FUNCTION_BLOCK Queue
VAR_INPUT
END_VAR
VAR_OUTPUT
END_VAR
VAR
	bAddTailValue		: BOOL := TRUE;
	bRemoveHeadValue	: BOOL := TRUE;
	bCount				: BOOL := TRUE;
	

END_VAR

END_FUNCTION_BLOCK

(* stored: Version 1.1.0.1, ProductVersion 3.1.4024.12
   POU Queue: Id {2b7de811-7be1-0bd1-2f1a-4b9eb91eca6a}, SpecialFunc None *)
